FUNCTION F_Sine : REAL
VAR_INPUT
	A		: REAL;	// Amplitude
	yoff	: REAL; // offset
	w		: REAL; // Kreisfrequenz (rad/s)
	t		: REAL; // Time (s)
END_VAR
VAR
END_VAR

F_Sine := (A * SIN(w*t)) + yoff;

END_FUNCTION

(* stored: Version 1.1.0.1, ProductVersion 3.1.4024.9
   POU F_Sine: Id {487d2d3b-3a85-4c4d-bc55-951ea6b2f182}, SpecialFunc None *)
